% RSLogix 500 project HOURMETER.RSS, saved by version 8.30.00.16 %
PROJECT "UNTITLED"    % processor: Bul.1763 MicroLogix 1100 Series B %

PROGRAM FILES
  LAD 2   10 rungs

DATA FILES
  O0 OUTPUT  5 elements
  I1 INPUT  7 elements
  S2 STATUS  66 elements
  B3 BINARY  1 elements
  T4 TIMER  4 elements
  C5 COUNTER  1 elements
  R6 CONTROL  1 elements
  N7 INTEGER  7 elements
  F8 FLOAT  1 elements

LADDER 2
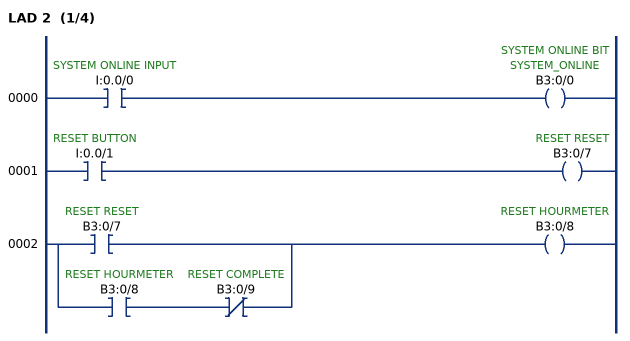
% Rung: 0 %
SOR XIC I:0.0/0 OTE B3:0/0 EOR
%   I:0.0/0  "SYSTEM ONLINE INPUT" %
%   B3:0/0  SYSTEM_ONLINE  "SYSTEM ONLINE BIT" %
% Rung: 1 %
SOR XIC I:0.0/1 OTE B3:0/7 EOR
%   I:0.0/1  "RESET BUTTON" %
%   B3:0/7  RESET  "RESET" %
% Rung: 2 %
SOR BST XIC B3:0/7 NXB XIC B3:0/8 XIO B3:0/9 BND OTE B3:0/8 EOR
%   B3:0/7  RESET  "RESET" %
%   B3:0/8  "RESET HOURMETER" %
%   B3:0/9  "RESET COMPLETE" %

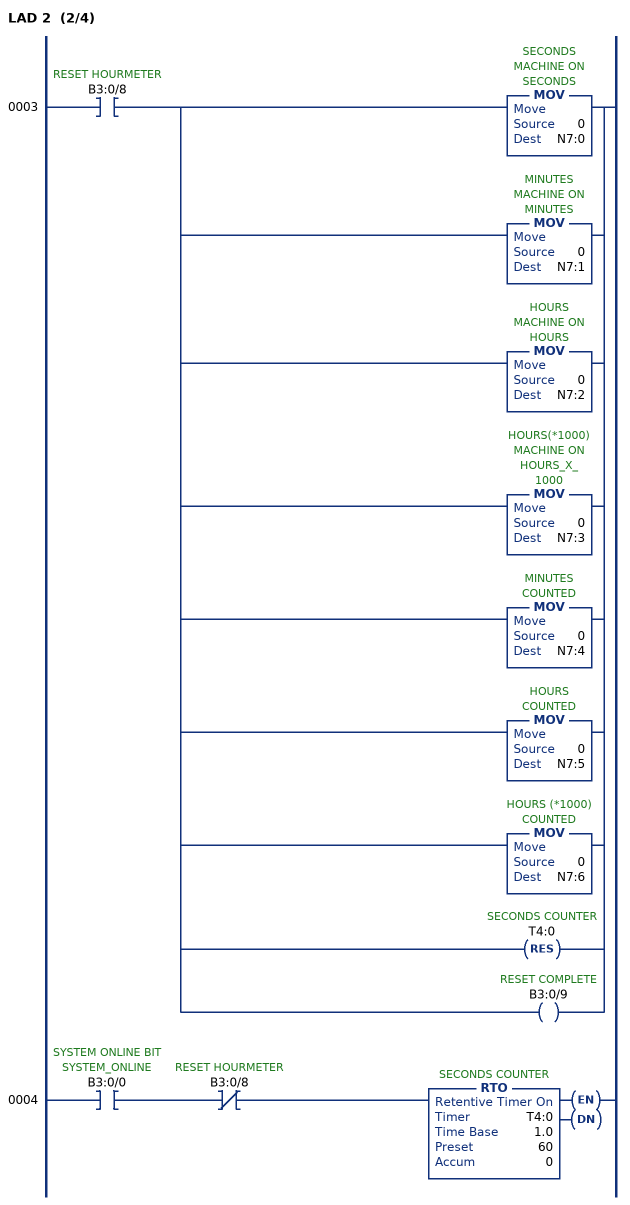
% Rung: 3 %
SOR XIC B3:0/8 BST MOV 0 N7:0 NXB MOV 0 N7:1 NXB MOV 0 N7:2 NXB MOV 0 N7:3 NXB MOV 0 N7:4 NXB MOV 0 N7:5 NXB MOV 0 N7:6 NXB RES T4:0 NXB OTE B3:0/9 BND EOR
%   B3:0/8  "RESET HOURMETER" %
%   N7:0  SECONDS  "SECONDS MACHINE ON" %
%   N7:1  MINUTES  "MINUTES MACHINE ON" %
%   N7:2  HOURS  "HOURS MACHINE ON" %
%   N7:3  HOURS_X_1000  "HOURS(*1000) MACHINE ON" %
%   N7:4  "MINUTES COUNTED" %
%   N7:5  "HOURS COUNTED" %
%   N7:6  "HOURS (*1000) COUNTED" %
%   T4:0  "SECONDS COUNTER" %
%   B3:0/9  "RESET COMPLETE" %
% Rung: 4 %
SOR XIC B3:0/0 XIO B3:0/8 RTO T4:0 1.0 60 0 EOR
%   B3:0/0  SYSTEM_ONLINE  "SYSTEM ONLINE BIT" %
%   B3:0/8  "RESET HOURMETER" %
%   T4:0  "SECONDS COUNTER" %

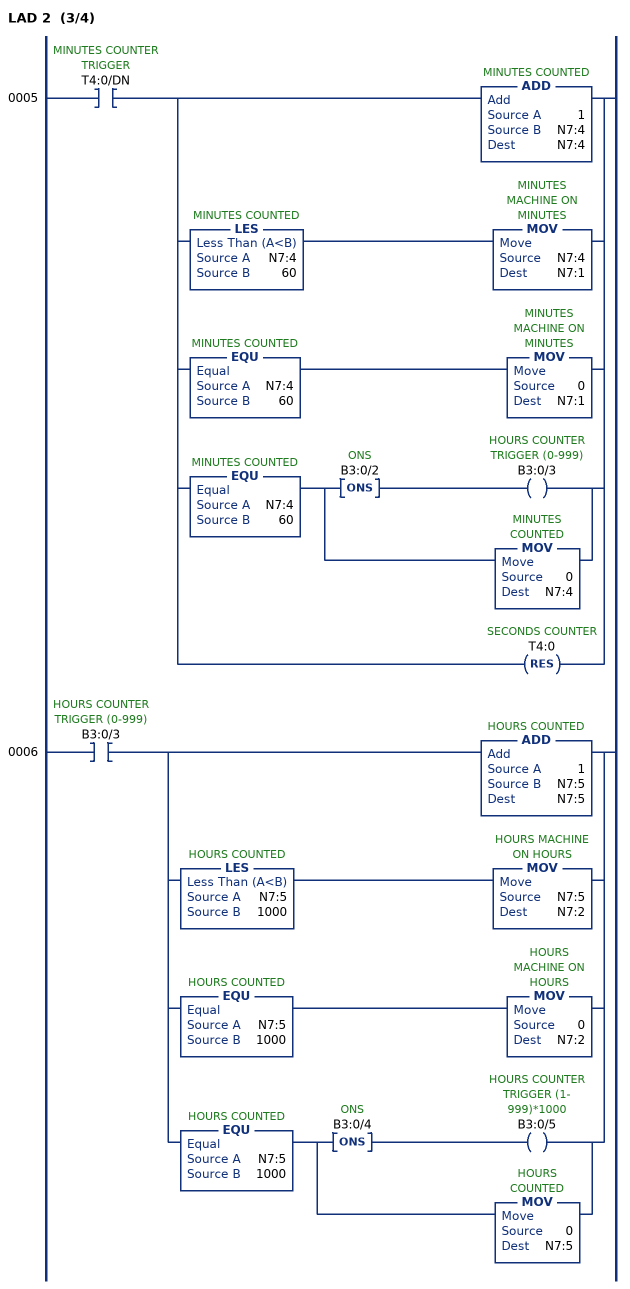
% Rung: 5 %
SOR XIC T4:0/DN BST ADD 1 N7:4 N7:4 NXB LES N7:4 60 MOV N7:4 N7:1 NXB EQU N7:4 60 MOV 0 N7:1 NXB EQU N7:4 60 BST ONS B3:0/2 OTE B3:0/3 NXB MOV 0 N7:4 BND NXB RES T4:0 BND EOR
%   T4:0/DN  "MINUTES COUNTER TRIGGER" %
%   N7:4  "MINUTES COUNTED" %
%   N7:1  MINUTES  "MINUTES MACHINE ON" %
%   B3:0/2  "ONS" %
%   B3:0/3  "HOURS COUNTER TRIGGER (0-999)" %
%   T4:0  "SECONDS COUNTER" %
% Rung: 6 %
SOR XIC B3:0/3 BST ADD 1 N7:5 N7:5 NXB LES N7:5 1000 MOV N7:5 N7:2 NXB EQU N7:5 1000 MOV 0 N7:2 NXB EQU N7:5 1000 BST ONS B3:0/4 OTE B3:0/5 NXB MOV 0 N7:5 BND BND EOR
%   B3:0/3  "HOURS COUNTER TRIGGER (0-999)" %
%   N7:5  "HOURS COUNTED" %
%   N7:2  HOURS  "HOURS MACHINE ON" %
%   B3:0/4  "ONS" %
%   B3:0/5  "HOURS COUNTER TRIGGER (1-999)*1000" %

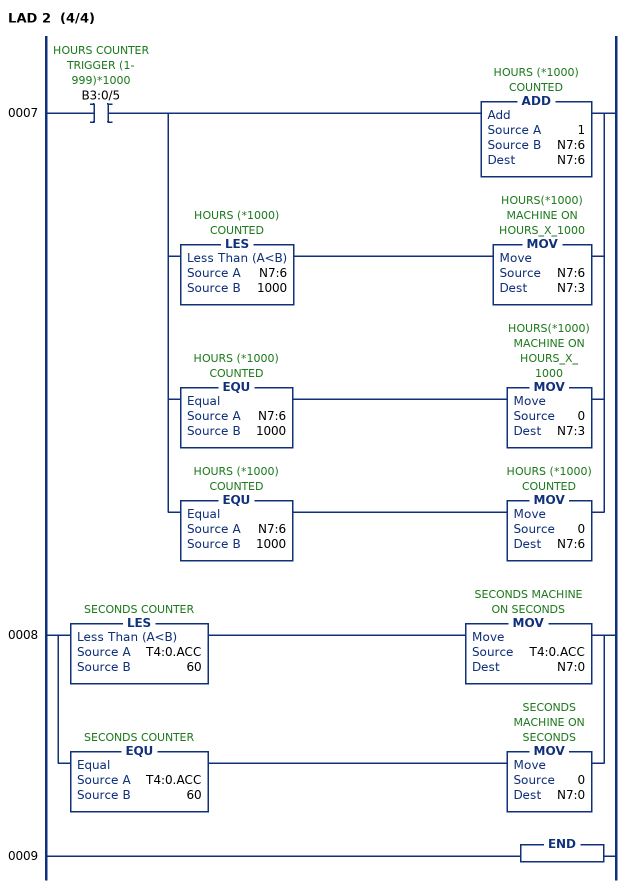
% Rung: 7 %
SOR XIC B3:0/5 BST ADD 1 N7:6 N7:6 NXB LES N7:6 1000 MOV N7:6 N7:3 NXB EQU N7:6 1000 MOV 0 N7:3 NXB EQU N7:6 1000 MOV 0 N7:6 BND EOR
%   B3:0/5  "HOURS COUNTER TRIGGER (1-999)*1000" %
%   N7:6  "HOURS (*1000) COUNTED" %
%   N7:3  HOURS_X_1000  "HOURS(*1000) MACHINE ON" %
% Rung: 8 %
SOR BST LES T4:0.ACC 60 MOV T4:0.ACC N7:0 NXB EQU T4:0.ACC 60 MOV 0 N7:0 BND EOR
%   T4:0  "SECONDS COUNTER" %
%   N7:0  SECONDS  "SECONDS MACHINE ON" %
% Rung: 9 %
SOR END EOR

OTHER DOCUMENTED ADDRESSES
  B3:0/1  "COUNTER START"
  B3:0/6  "ONS"
  C5:0  "SECONDS COUNTER"
  T4:1  "MINUTES COUNTER"
  T4:1/DN  "HOURS COUNTER TRIGGER (0-999)"
  T4:2  "HOURS COUNTER (0- 999)"
  T4:2/DN  "HOURS COUNTER TRIGGER (1-999)*1000"
  T4:3  "HOURS COUNTER (1- 999)*1000"

DATA TABLE (non-zero values as saved)
DATA T4
% .PRE .ACC %
% T4:0 % 60 0
% T4:1 % 60 0
% T4:2 % 1000 0
% T4:3 % 1000 0
